FUNCTION_BLOCK FB_Xbox_Controller
VAR
	{attribute 'hide'}
	_AmsNetId : T_AMSNETID;
	{attribute 'hide'}
	_WriteServerData : ADSWRITE;
	{attribute 'hide'}
	_ReadServerData : ADSREAD;
	// RAW ADS Inputs for debug (Use properties to access items)
	stXboxControllerInputs : ST_Xbox_Controller_ADS_Inputs;
	{attribute 'hide'}
	_stRumble : ST_Xbox_Controller_Rumble;
	{attribute 'hide'}
	_IDXGRP : UDINT;
	{attribute 'hide'}
	_rumbleCommand 			: ST_Xbox_Class_Command_Status;
	{attribute 'hide'}
	_stControllerButtons 	: ST_Xbox_Controller_Buttons;
	{attribute 'hide'}
	_stControllerStatus		: ST_Xbox_Controller_Status;
	{attribute 'hide'}
	_stLeftJoystick 		: ST_Xbox_Controller_Joystick;
	{attribute 'hide'}
	_stRightJoystick 		: ST_Xbox_Controller_Joystick;
	{attribute 'hide'}
	_fLeftTrigger 			: REAL;
	{attribute 'hide'}
	_fRightTrigger 			: REAL;
	{attribute 'hide'}
	_bSetRumbleEvent 		: BOOL; // Internal indication of an ADS write event
	{attribute 'hide'}
	_bSetRumbleEventLogged	: BOOL; // Check if the Set Rumble event is being called too many times	
END_VAR

// This method is called cyclically to update the controller inputs
METHOD Cycle : BOOL
// Read the current inputs
THIS^._ReadServerData(
	NETID:= THIS^._AmsNetId, 
	PORT:= 25733, 
	IDXGRP:= THIS^._IDXGRP, 
	IDXOFFS:= 0, 
	LEN:= SIZEOF(THIS^.stXboxControllerInputs), 
	DESTADDR:= ADR(THIS^.stXboxControllerInputs), 
	READ:= TRUE, 
	TMOUT:= T#5S,
	ERR=>);
	
// If there is an error in reading from the server, shut all inputs off
IF THIS^._ReadServerData.ERR THEN
	memset(ADR(THIS^.stXboxControllerInputs), 0, SIZEOF(THIS^.stXboxControllerInputs));
END_IF

// Stop read command
THIS^._ReadServerData(
	NETID:= THIS^._AmsNetId, 
	PORT:= 25733, 
	IDXGRP:= THIS^._IDXGRP, 
	IDXOFFS:= 0, 
	LEN:= SIZEOF(THIS^.stXboxControllerInputs), 
	DESTADDR:= ADR(THIS^.stXboxControllerInputs), 
	READ:= FALSE, 
	TMOUT:= T#5S,
	ERR=>);
	

// Handle any write requests for the rumble
// Write the new values
THIS^._WriteServerData(
	NETID:= THIS^._AmsNetId, 
	PORT:= 25733, 
	IDXGRP:= THIS^._IDXGRP, 
	IDXOFFS:= 16, 
	LEN:= SIZEOF(THIS^._stRumble), 
	SRCADDR:= ADR(THIS^._stRumble), 
	WRITE:= THIS^._bSetRumbleEvent, 
	TMOUT:= T#5S);
	
// Update the status of the current command if active
IF 	THIS^._bSetRumbleEvent THEN
	THIS^.P_SetRumble.bBusy := THIS^._WriteServerData.BUSY;
	THIS^.P_SetRumble.bError := THIS^._WriteServerData.ERR;
END_IF

// Check if it's done writing
IF THIS^._bSetRumbleEvent AND NOT THIS^._WriteServerData.BUSY THEN
	IF NOT THIS^._WriteServerData.ERR THEN
		THIS^.P_SetRumble.bDone := TRUE;
	END_IF
	// Turn off the write request
	THIS^._WriteServerData(
		NETID:= THIS^._AmsNetId, 
		PORT:= 25733, 
		IDXGRP:= THIS^._IDXGRP, 
		IDXOFFS:= 16, 
		LEN:= SIZEOF(THIS^._stRumble), 
		SRCADDR:= ADR(THIS^._stRumble), 
		WRITE:= FALSE, 
		TMOUT:= T#5S);
		
	THIS^._bSetRumbleEvent := FALSE;
END_IF
END_METHOD

METHOD FB_init : BOOL
VAR_INPUT
	bInitRetains : BOOL; // if TRUE, the retain variables are initialized (warm start / cold start)
	bInCopyCode : BOOL;  // if TRUE, the instance afterwards gets moved into the copy code (online change)
	NetID 				: T_AMSNETID := ''; // AMS Net ID of the Xbox Service Provider
	iControllerNumber 	: UINT(1..4) := 1; // The controller number for the controller you'd like to use
END_VAR
THIS^._AmsNetId := NetID;
THIS^._IDXGRP := iControllerNumber * 16#10000;
END_METHOD

{attribute 'monitoring':='call'}
// Structure of the different active buttons
PROPERTY P_Buttons : REFERENCE TO ST_Xbox_Controller_Buttons
GET
IF THIS^.stXboxControllerInputs.bStatus.xConnected THEN	
	THIS^._stControllerButtons.DPad.bUp				:= THIS^.stXboxControllerInputs.bButtons.xDPAD_UP;
	THIS^._stControllerButtons.DPad.bDown			:= THIS^.stXboxControllerInputs.bButtons.xDPAD_DOWN;
	THIS^._stControllerButtons.DPad.bLeft			:= THIS^.stXboxControllerInputs.bButtons.xDPAD_LEFT;
	THIS^._stControllerButtons.DPad.bRight			:= THIS^.stXboxControllerInputs.bButtons.xDPAD_RIGHT;
	THIS^._stControllerButtons.bStart  				:= THIS^.stXboxControllerInputs.bButtons.xSTART;
	THIS^._stControllerButtons.bBack  				:= THIS^.stXboxControllerInputs.bButtons.xBACK;
	THIS^._stControllerButtons.bLeft_Thumbstick  	:= THIS^.stXboxControllerInputs.bButtons.xLEFT_THUMB;
	THIS^._stControllerButtons.bRight_Thumbstick 	:= THIS^.stXboxControllerInputs.bButtons.xRIGHT_THUMB;
	THIS^._stControllerButtons.bLeft_Shoulder  		:= THIS^.stXboxControllerInputs.bButtons.xLEFT_SHOULDER;
	THIS^._stControllerButtons.bRight_Shoulder  	:= THIS^.stXboxControllerInputs.bButtons.xRIGHT_SHOULDER;
	THIS^._stControllerButtons.bA_Button  			:= THIS^.stXboxControllerInputs.bButtons.xA;
	THIS^._stControllerButtons.bB_Button  			:= THIS^.stXboxControllerInputs.bButtons.xB;
	THIS^._stControllerButtons.bX_Button  			:= THIS^.stXboxControllerInputs.bButtons.xX;
	THIS^._stControllerButtons.bY_Button  			:= THIS^.stXboxControllerInputs.bButtons.xY;
ELSE
	THIS^._stControllerButtons.DPad.bUp				:= FALSE;
	THIS^._stControllerButtons.DPad.bDown			:= FALSE;
	THIS^._stControllerButtons.DPad.bLeft			:= FALSE;
	THIS^._stControllerButtons.DPad.bRight			:= FALSE;
	THIS^._stControllerButtons.bStart  				:= FALSE;
	THIS^._stControllerButtons.bBack  				:= FALSE;
	THIS^._stControllerButtons.bLeft_Thumbstick  	:= FALSE;
	THIS^._stControllerButtons.bRight_Thumbstick 	:= FALSE;
	THIS^._stControllerButtons.bLeft_Shoulder  		:= FALSE;
	THIS^._stControllerButtons.bRight_Shoulder  	:= FALSE;
	THIS^._stControllerButtons.bA_Button  			:= FALSE;
	THIS^._stControllerButtons.bB_Button  			:= FALSE;
	THIS^._stControllerButtons.bX_Button  			:= FALSE;
	THIS^._stControllerButtons.bY_Button  			:= FALSE;
END_IF
P_Buttons REF= THIS^._stControllerButtons;
END_GET
END_PROPERTY

{attribute 'monitoring':='call'}
// Returns a structure of data for the XY Joystick values
PROPERTY P_Left_Joystick : REFERENCE TO ST_Xbox_Controller_Joystick
GET
IF THIS^.stXboxControllerInputs.bStatus.xConnected THEN	
	THIS^._stLeftJoystick.fX := THIS^.stXboxControllerInputs.stLeft_Joystick.fX;
	THIS^._stLeftJoystick.fY := THIS^.stXboxControllerInputs.stLeft_Joystick.fY;
ELSE
	THIS^._stLeftJoystick.fX := 0;
	THIS^._stLeftJoystick.fY := 0;
END_IF
P_Left_Joystick REF= THIS^._stLeftJoystick;
END_GET
END_PROPERTY

{attribute 'monitoring':='call'}
// Left trigger value
PROPERTY P_Left_Trigger : REFERENCE TO REAL
GET
IF THIS^.stXboxControllerInputs.bStatus.xConnected THEN	
	THIS^._fLeftTrigger := THIS^.stXboxControllerInputs.fLeft_Trigger;
ELSE
	THIS^._fLeftTrigger := 0;
END_IF
P_Left_Trigger REF= THIS^._fLeftTrigger;
END_GET
END_PROPERTY

{attribute 'monitoring':='call'}
// Returns a structure of data for the XY Joystick values
PROPERTY P_Right_Joystick : REFERENCE TO ST_Xbox_Controller_Joystick
GET
IF THIS^.stXboxControllerInputs.bStatus.xConnected THEN	
	THIS^._stRightJoystick.fX := THIS^.stXboxControllerInputs.stRight_Joystick.fX;
	THIS^._stRightJoystick.fY := THIS^.stXboxControllerInputs.stRight_Joystick.fY;
ELSE
	THIS^._stRightJoystick.fX := 0;
	THIS^._stRightJoystick.fY := 0;
END_IF
P_Right_Joystick REF= THIS^._stRightJoystick;
END_GET
END_PROPERTY

{attribute 'monitoring':='call'}
// Right trigger value
PROPERTY P_Right_Trigger : REFERENCE TO REAL
GET
IF THIS^.stXboxControllerInputs.bStatus.xConnected THEN	
	THIS^._fRightTrigger := THIS^.stXboxControllerInputs.fRight_Trigger;
ELSE
	THIS^._fRightTrigger := 0;
END_IF
P_Right_Trigger REF= THIS^._fRightTrigger;
END_GET
END_PROPERTY

{attribute 'monitoring':='call'}
// Status of the SetRumble method
PROPERTY P_SetRumble : REFERENCE TO ST_Xbox_Class_Command_Status
GET
P_SetRumble REF= THIS^._rumbleCommand;
END_GET
END_PROPERTY

{attribute 'monitoring':='call'}
// Structure of the controller capabilites and status
PROPERTY P_Status : REFERENCE TO ST_Xbox_Controller_Status
GET
IF THIS^.stXboxControllerInputs.bStatus.xConnected THEN	
	THIS^._stControllerStatus.bConnected 		:= TRUE;
	THIS^._stControllerStatus.bDisconnected 	:= FALSE;
	THIS^._stControllerStatus.iControllerNumber := THIS^.stXboxControllerInputs.iControllerNumber;
ELSE
	THIS^._stControllerStatus.bConnected 		:= FALSE;
	THIS^._stControllerStatus.bDisconnected 	:= TRUE;
	THIS^._stControllerStatus.iControllerNumber := 0;
END_IF

IF THIS^.stXboxControllerInputs.bStatus.xBattery_Type_Disconnected THEN
	THIS^._stControllerStatus.eBattery_Type := E_Xbox_Controller_Battery_Types.Disconnected;
END_IF

IF THIS^.stXboxControllerInputs.bStatus.xBattery_Type_Wired THEN
	THIS^._stControllerStatus.eBattery_Type := E_Xbox_Controller_Battery_Types.Wired;
END_IF

IF THIS^.stXboxControllerInputs.bStatus.xBattery_Type_Alkaline THEN
	THIS^._stControllerStatus.eBattery_Type := E_Xbox_Controller_Battery_Types.Alkaline;
END_IF

IF THIS^.stXboxControllerInputs.bStatus.xBattery_Type_NIMH THEN
	THIS^._stControllerStatus.eBattery_Type := E_Xbox_Controller_Battery_Types.NIMH;
END_IF

IF THIS^.stXboxControllerInputs.bStatus.xBattery_Type_Unknown THEN
	THIS^._stControllerStatus.eBattery_Type := E_Xbox_Controller_Battery_Types.Unknown;
END_IF

IF THIS^.stXboxControllerInputs.bStatus.xBattery_Level_Empty THEN
	THIS^._stControllerStatus.eBattery_Level := E_Xbox_Controller_Battery_Levels.Empty;
END_IF

IF THIS^.stXboxControllerInputs.bStatus.xBattery_Level_Low THEN
	THIS^._stControllerStatus.eBattery_Level := E_Xbox_Controller_Battery_Levels.Low;
END_IF

IF THIS^.stXboxControllerInputs.bStatus.xBattery_Level_Medium THEN
	THIS^._stControllerStatus.eBattery_Level := E_Xbox_Controller_Battery_Levels.Medium;
END_IF

IF THIS^.stXboxControllerInputs.bStatus.xBattery_Level_Full THEN
	THIS^._stControllerStatus.eBattery_Level := E_Xbox_Controller_Battery_Levels.Full;
END_IF


P_Status REF= THIS^._stControllerStatus;
END_GET
END_PROPERTY

// Sets the rumble for the controller
METHOD SetRumble : BOOL
VAR_INPUT
	// Left motor speed (0..100%)
	fLeftMotor : REAL;
	// Right motor speed (0..100%)
	fRightMotor : REAL;
END_VAR
// When the method is called, check if a write is in progress
IF THIS^._bSetRumbleEvent THEN
	// ADS you are doing that too much
	IF NOT THIS^._bSetRumbleEventLogged THEN
		ADSLOGSTR( msgCtrlMask := ADSLOG_MSGTYPE_WARN, msgFmtStr := 'PLC Msg.: Command being called too often, wait for done bit: %s', strArg := 'SetRumble()');
		THIS^._bSetRumbleEventLogged := TRUE;
	END_IF	
ELSE
	// Check if the value is within range
	IF fLeftMotor > 100 THEN
		THIS^._stRumble.fLeftMotor := 100.0;
	ELSIF fLeftMotor < 0 THEN
		THIS^._stRumble.fLeftMotor := 0.0;
	ELSE
		THIS^._stRumble.fLeftMotor := fLeftMotor;
	END_IF
	
	// Check if the value is within range
	IF fRightMotor > 100 THEN
		THIS^._stRumble.fRightMotor := 100.0;
	ELSIF fRightMotor < 0 THEN
		THIS^._stRumble.fRightMotor := 0.0;
	ELSE
		THIS^._stRumble.fRightMotor := fRightMotor;
	END_IF
	
	//Reset all status for the command
	THIS^.P_SetRumble.bDone := FALSE;
	THIS^.P_SetRumble.bBusy := FALSE;
	THIS^.P_SetRumble.bError := FALSE;

	// Set the high bit on the write command
	THIS^._bSetRumbleEvent := TRUE;
END_IF

// If it's done, set the current even in progress to false
IF P_SetRumble.bDone THEN
	THIS^._bSetRumbleEvent := FALSE;
END_IF

// Event Received
SetRumble := THIS^._bSetRumbleEvent;
END_METHOD

END_FUNCTION_BLOCK

(* stored: Version 1.1.0.1, ProductVersion 3.1.4024.11
   POU FB_Xbox_Controller: Id {16e61ff8-1d18-479b-8b07-5a4f238667a6}, SpecialFunc None
   Method Cycle: Id {c4c654fa-155e-401b-8a85-1aefc3ab660f}
   Method FB_init: Id {5ca1819e-d48f-4374-9f4b-b509d7da22ed}
   Property P_Buttons: Id {9ecee726-55c8-4ab8-9170-a864e7a68da5}
   Get Get: Id {fabea6d4-f972-48bb-9b75-17006ffd152b}
   Property P_Left_Joystick: Id {33db2771-a51a-47cd-87e9-82222a82ae74}
   Get Get: Id {4b140f7b-8969-4350-962e-103fcb9f7ed9}
   Property P_Left_Trigger: Id {4760222a-9195-417e-97df-e345197e8a07}
   Get Get: Id {1906a11d-9ff5-4e03-b10e-492065686575}
   Property P_Right_Joystick: Id {e8db0053-5241-40a3-8cab-5544d5c2006b}
   Get Get: Id {0e92480b-9055-499c-897c-becbad0c9d16}
   Property P_Right_Trigger: Id {78732f9d-af31-4e4c-821e-1f8189aa19ee}
   Get Get: Id {f85af2b8-09ba-4400-a23b-f2e4aab2e32c}
   Property P_SetRumble: Id {e951a137-f153-4333-bf9b-6c5d979a71f2}
   Get Get: Id {1009e700-d671-4ebf-b638-5a140a7d5a04}
   Property P_Status: Id {9862bf27-d17e-48b2-b703-c886caf0e3f2}
   Get Get: Id {dabe201a-2054-48fe-a490-6ba481e4db51}
   Method SetRumble: Id {321f1c4d-4b89-4b24-88d5-c2d524fc2f0a} *)
